TYPE csp_case_flap_control_phase_status_enum :
(		
	CSP_CASE_FLAP_CONTROL_STATUS_PHASE_START							:= 0,
	CSP_CASE_FLAP_CONTROL_STATUS_PHASE_DISABLE 							:= 10,
	CSP_CASE_FLAP_CONTROL_STATUS_PHASE_ENABLE 							:= 20,	
	CSP_CASE_FLAP_CONTROL_STATUS_PHASE_ENABLED 							:= 30,
	CSP_CASE_FLAP_CONTROL_STATUS_PHASE_CALCULATE_SLAVE_POSITION_REQUEST	:= 31,
	CSP_CASE_FLAP_CONTROL_STATUS_PHASE_CALCULATING_SLAVE_POSITION		:= 32,
	CSP_CASE_FLAP_CONTROL_STATUS_PHASE_REQUESTED						:= 33,
	CSP_CASE_FLAP_CONTROL_STATUS_PHASE_PHASING							:= 34,
	CSP_CASE_FLAP_CONTROL_STATUS_PHASE_PHASED							:= 35,
	CSP_CASE_FLAP_CONTROL_STATUS_PHASE_REDEFINE							:= 40,
	CSP_CASE_FLAP_CONTROL_STATUS_PHASE_REDEFINED						:= 50,
	CSP_CASE_FLAP_CONTROL_STATUS_PHASE_DONE 							:= 900,
	CSP_CASE_FLAP_CONTROL_STATUS_PHASE_ERROR 							:= 999
) := CSP_CASE_FLAP_CONTROL_STATUS_PHASE_START;
END_TYPE

(* stored: Version 1.1.0.1, ProductVersion 3.1.4024.3
   DUT csp_case_flap_control_phase_status_enum: Id {cb136916-23eb-0d9a-0521-bb17fbdb6193} *)
